{attribute 'OPC.UA.DA' := '1'}
{attribute 'OPC.UA.DA.StructuredType' := '1'}
TYPE AttenuationMsg :
STRUCT
	Id : EPowerIlluminationFlow;
	Attenuation : UINT;
END_STRUCT
END_TYPE

(* stored: Version 1.1.0.1, ProductVersion 3.1.4024.10
   DUT AttenuationMsg: Id {16b8a0e2-d5cf-43a6-ace1-a7017d2031de} *)
